FUNCTION Convert_TOD_TO_BOOL : BOOL
VAR_INPUT
	in : TOD;
	out : REFERENCE TO BOOL;
END_VAR
VAR
	converted : BOOL;
END_VAR

converted := TOD_TO_BOOL(in);

IF (BOOL_TO_TOD(converted) <> in) THEN
	RETURN;
END_IF

out := converted;
Convert_TOD_TO_BOOL := TRUE;

END_FUNCTION

(* stored: Version 1.1.0.1, ProductVersion 3.1.4024.12
   POU Convert_TOD_TO_BOOL: Id {8db8181b-67df-4fe1-9a35-85875558dd97}, SpecialFunc None *)
